// Usage:
// Call instance (i.e. ofbCsvRead();) every scan while waiting for operations to complete.
// SetFileParams() Set the File directory and separator variable. 
// GetFile() Get the File.
// #various props: Observe the properties to see whether it passed the file checks.
// NextField() Next through the fields of the CSV. 
// #sField, Row, Column: Use properties to access values, using row and column.
FUNCTION_BLOCK T_CsvFileWriter
VAR
// state vars.
	filePath : Tc2_Utilities.T_MaxString; // filepath
	
// backing properties	
	_Row : UINT; // current Row number (zero indexed)
	_Column : UINT; // current Column number (zero indexed)
	_Error : BOOL;
	_ErrorId : UDINT; // E_AdsErr
	
// Objects	
	fileWrite : T_FileWriteBase;(* Writes one record (line) *)
	
END_VAR

fileWrite();

METHOD PUBLIC AddStringField// Add Field. Adds CSV separator to previous field, if it exists
VAR_INPUT 
	sFieldString : STRING; 
END_VAR

VAR_INST
	sFieldStringLocal : STRING; // This has a valid memory address (inputs dont)
END_VAR
sFieldStringLocal := sFieldString;
// append separator to previous field if not first field
IF _Column > 0 THEN 
	
	fileWrite.AppendToBuffer(
		pDataForBuffer := ADR(Tc2_Utilities.DEFAULT_CSV_FIELD_SEP),
		DataLength := SIZEOF(Tc2_Utilities.DEFAULT_CSV_FIELD_SEP)
	);	

	IF Error THEN // Error looks at FileWrite.Error
		RETURN;
	END_IF
	
END_IF

// Add string.
fileWrite.AppendToBuffer(
	pDataForBuffer := ADR(sFieldStringLocal),
	DataLength := INT_TO_UDINT(LEN(sFieldString))
);

IF Error THEN // Error looks at FileWrite.Error
	RETURN;
END_IF

_Column := _Column + 1;
END_METHOD

{attribute 'monitoring' := 'call'}
PROPERTY PUBLIC BufferClear : BOOL // ready for first entry after ResetWriteBuffer
GET
BufferClear := fileWrite.BufferClear;
END_GET
END_PROPERTY

{attribute 'monitoring' := 'call'}
PROPERTY PUBLIC Busy : BOOL
GET
Busy := fileWrite.Busy;
END_GET
END_PROPERTY

METHOD PUBLIC ClearBuffer : BOOL // Clears the buffer for first write.
ClearBuffer := fileWrite.ClearWriteBuffer();
_Error := fileWrite.Error;
_ErrorId := fileWrite.ErrorId;

_Column := 0;
_Row := 0;
END_METHOD

PROPERTY PUBLIC Column : UINT
GET
Column := _Column;
END_GET
END_PROPERTY

{attribute 'monitoring' := 'call'}
PROPERTY PUBLIC Done : BOOL
GET
Done := fileWrite.Done;
END_GET
END_PROPERTY

{attribute 'monitoring' := 'call'}
PROPERTY PUBLIC Error : BOOL
GET
_Error := fileWrite.Error;
Error := _Error;
END_GET
END_PROPERTY

{attribute 'monitoring' := 'call'}
PROPERTY PUBLIC ErrorId : UDINT
GET
_ErrorId := fileWrite.ErrorId;
ErrorId := _ErrorId;
END_GET
END_PROPERTY

METHOD PUBLIC NewLine // Make a New Line in the File
VAR_INST
	tempByte : BYTE;
END_VAR
VAR CONSTANT
	CARRIAGE_RETURN : BYTE := 16#D;
	LINE_FEED : BYTE := 16#A;
END_VAR
// load up CR.
tempByte := CARRIAGE_RETURN;

//Write.
fileWrite.AppendToBuffer(
		pDataForBuffer := ADR(tempByte),
		DataLength := SIZEOF(tempByte)
	);

// check for errors
IF Error THEN // Error looks at FileWrite.Error
	RETURN;
END_IF

// load up LF.
tempByte := LINE_FEED;

//Write.
fileWrite.AppendToBuffer(
		pDataForBuffer := ADR(tempByte),
		DataLength := SIZEOF(tempByte)
	);	

// check for errors
IF Error THEN // Error looks at FileWrite.Error
	RETURN;
END_IF

_Row := _Row + 1;
_Column := 0;
END_METHOD

PROPERTY PUBLIC Row : UINT
GET
Row := _Row;
END_GET
END_PROPERTY

METHOD PUBLIC SetFileParams
VAR_INPUT
	FilePath : Tc2_Utilities.T_MaxString;
	Separator: BYTE; // Updates TC Utilities Global_Variables DEFAULT_CSV_FIELD_SEP
END_VAR
VAR_INST
	debugCount : INT;
END_VAR
VAR CONSTANT
	ASCI_SEMI_COLON : BYTE := 16#3B;
	ASCI_COMMA		: BYTE := 16#2C;
END_VAR
// THIS^ references the base object properties
THIS^.filePath := FilePath; // for debug only.

fileWrite.SetFilePath(FilePath := FilePath);

// Validate separator.
IF Separator = ASCI_SEMI_COLON THEN
	Tc2_Utilities.DEFAULT_CSV_FIELD_SEP := 16#3B;
	
ELSIF Separator = ASCI_COMMA THEN
	Tc2_Utilities.DEFAULT_CSV_FIELD_SEP := 16#3B;
	
ELSE
	Tc2_Utilities.DEFAULT_CSV_FIELD_SEP := 16#3B;
	
END_IF

debugCount := debugCount + 1;
END_METHOD

METHOD PUBLIC WriteToFile // Write Buffer to File. Calls "NewLine"() first.
IF Error THEN // Error looks at FileWrite.Error
	RETURN;
END_IF

// always add final CRLF.
NewLine();

IF Error THEN // Error looks at FileWrite.Error
	RETURN;
END_IF

fileWrite.StartWrite();
END_METHOD

END_FUNCTION_BLOCK

(* stored: Version 1.1.0.1, ProductVersion 3.1.4022.12
   POU T_CsvFileWriter: Id {1085c9eb-e997-446a-b003-e836d48add8e}, SpecialFunc None
   Folder Methods: Id {851d5649-a418-4459-be3f-e02c0e797249}
   Folder Properties: Id {b659b1b2-9be8-4a5a-ae17-3f1cba8e2b83}
   Method AddStringField: Id {6b256194-708f-47b4-8712-19db3b00ab17}
   Property BufferClear: Id {901fb2e9-30b2-48f5-b584-516e533e298f}
   Get Get: Id {87d640a3-c412-4888-b13f-b0c746de5570}
   Property Busy: Id {41c6db38-0b0d-4447-b64b-3e8adc0e26f7}
   Get Get: Id {f2505e27-9442-4b46-8e12-aa93326ad056}
   Method ClearBuffer: Id {5cf7386f-4069-47c8-8b51-3c7915ff54c3}
   Property Column: Id {4154d437-670b-4c46-8189-dec07219bf56}
   Get Get: Id {5229104c-11a4-430e-b480-93838f039e95}
   Property Done: Id {d42f7110-5897-439c-bbae-068242a89b8f}
   Get Get: Id {659f3dc4-56a5-4e91-9c8b-70c7354c677e}
   Property Error: Id {cabe518f-7a20-4f3b-af75-f0b5fd981f35}
   Get Get: Id {2e30b962-2af5-4d3a-aa4f-b94fffa0c7f3}
   Property ErrorId: Id {8a0ad82f-2047-407f-be26-a8a4d373d613}
   Get Get: Id {af85b4d7-6517-4d60-b88b-9b3abd8c09df}
   Method NewLine: Id {098e0aae-9b88-4db9-b422-7efa6a9d491f}
   Property Row: Id {b6894911-a846-43d5-8a56-942db9a3d87a}
   Get Get: Id {02c22d10-04b0-4b99-a2c8-c214c28f1c74}
   Method SetFileParams: Id {6d2c1a3e-b8ca-4bf4-a258-44ae4a711c36}
   Method WriteToFile: Id {52b0a0ab-c039-44db-b778-31b0420765df} *)
